PROGRAM MAIN
VAR
	heartbeat : BYTE;
	out1 AT %Q* : BOOL;
	outVal1 : BOOL;
END_VAR

VARS.iSum := VARS.iTest1 + VARS.iTest2 + 10;
//heartbeat:= heartbeat+1;
out1 := outval1;

END_PROGRAM

(* stored: Version 1.1.0.1, ProductVersion 3.1.4022.12
   POU MAIN: Id {cf6af052-128c-45b0-b894-0c0872c9da64}, SpecialFunc None *)
